// TwinCAT 3 PLC project Projekt
// ProgramVersion: 3.1.4023.0
// libraries:
//   Tc2_MC2, * (Beckhoff Automation GmbH)
//   Tc2_MC2_Camming, * (Beckhoff Automation GmbH)
//   Tc2_MC2_Drive, * (Beckhoff Automation GmbH)
//   Tc2_Standard, * (Beckhoff Automation GmbH)
//   Tc2_System, * (Beckhoff Automation GmbH)
//   Tc2_Utilities, * (Beckhoff Automation GmbH)
//   Tc3_Module, * (Beckhoff Automation GmbH)
// project tree:
//   GVLs/ IO.TcGVL
//   / PlcTask.TcTTO (not stored)
//   POUs/ FB_INICIALIZACIJA.TcPOU, MAIN.TcPOU, PRG_INIT.TcPOU
// real-time tasks:
//   TASK PlcTask: cycle T#10ms, priority 20, ADS port 350
// motion (NC):
//   TASK NC-Task 1 SAF: cycle T#2ms, priority 4, ADS port 501
//   TASK NC-Task 1 SVB: cycle T#10ms, priority 8, ADS port 511
//   AXIS SLAVE - AX5000 (id 1)
//     General: UnitName=°
//     Dynamic: Acceleration=5029.17, Deceleration=5029.17, Jerk=651703
//     Velo: RefSearch=38.8099189453125, RefSync=38.8099189453125, SlowManual=194.049594726563, FastManual=1164.29756835938, Fast=3880.99189453125, Maximum=3880.99
//     PositionAreaControl: Enable=false
//     TargetPosControl: Enable=false
//     OtherSettings: AllowMotionCmdToSlave=true
//     encoder EncType=8
//       EncPara: ScaleFactorNumerator=36, ScaleFactorDenominator=1048576, MaxCount=#xffffffff
//         Inc: RefSearchInverse=true, RefSyncInverse=false
//         TimeComp: TimeCompMode=1, EncDelayCycles=4
//     drive DrvType=9
//       DrvPara: MaxCount=#xffffffff, DriveControlDWord=#x00030100
//         Analog: VeloReferenz=4269.09108398438, VeloScale=1.02400649589962, TorqueSetpointScale=10, ScaleFactorActTorque=0.1
//         TimeComp: TaskDelayCycles=1
//     controller CtrType=1
//       CtrPara: PriorControlFactor=1
//         PosDiffControl: Enable=false
//         Observer: BandWidth=20
//   AXIS Enkoder_Axis (id 2)
//     General: UnitName=°, UnitFlags=#x00000004
//     Dynamic: AccelerationMaximum=25000, DecelerationMaximum=25000
//     Velo: Maximum=20000
//     PositionAreaControl: Enable=false
//     TargetPosControl: Enable=false
//     OtherSettings: AllowMotionCmdToSlave=true
//     encoder EncType=4
//       EncPara: ScaleFactorNumerator=1, MaxCount=#xffffffff
//         Inc: RefSoftSyncMask=#x0000ffff
//     drive DrvType=5
//       Analog: VeloReferenz=22000, TorqueSetpointScale=10, ScaleFactorActTorque=0.1
//       TimeComp: TaskDelayCycles=1
//     controller CtrType=1
//       CtrPara: PriorControlFactor=1
//         PosDiffControl: Enable=false
//         Observer: BandWidth=20
//   AXIS Axis 3 (id 3)
//     OtherSettings: AllowMotionCmdToSlave=true
//     encoder EncType=1
//     drive DrvType=5
//       Analog: TorqueSetpointScale=10, ScaleFactorActTorque=0.1
//       TimeComp: TaskDelayCycles=1
//     controller CtrType=1
//       CtrPara: PriorControlFactor=1
//         Observer: BandWidth=20
//   AXIS Axis 4 HENGSTLER (id 4)
//     General: UnitName=°, UnitFlags=#x00000004
//     OtherSettings: AllowMotionCmdToSlave=true
//     encoder EncType=5
//       EncPara: ScaleFactorNumerator=360, ScaleFactorDenominator=4096, ReferenceSystem=1
//     drive DrvType=5
//       Analog: TorqueSetpointScale=10, ScaleFactorActTorque=0.1
//       TimeComp: TaskDelayCycles=1
//     controller CtrType=1
//       CtrPara: PriorControlFactor=1
//         Observer: BandWidth=20
// I/O:
//   DEVICE Device 1 (EtherCAT), AmsNetId 5.67.218.26.2.1
//     Term 10 (EK1200) [EK1200-5000 EtherCAT Power supply (2A E-Bus)]
//       Term 10 (EL2252) [EL2252 2Ch. Dig. Output 24V, 0.5A, DC Time Stamp]
//       Term 11 (EL1252) [EL1252 2Ch. Fast Dig. Input 24V, 1µs, DC Latch]
//       Term 12 (EL2004) [EL2004 4Ch. Dig. Output 24V, 0.5A]
//       Term 13 (EL2004) [EL2004 4Ch. Dig. Output 24V, 0.5A]
//       Term 14 (EL1014) [EL1014 4Ch. Dig. Input 24V, 10µs]
//       Term 15 (EL5151-0021) [EL5151-0021 1Ch. Inc. Encoder, 24V DC Output]
//       Term 1 (EL5001) [EL5001 1Ch. SSI Encoder]
//       Term 17 (EL9011) [EL9011 End Terminal]
//   DEVICE Device 4 (EtherCAT), AmsNetId 5.67.218.26.5.1
//     Drive 8 (AX5106-0000-0214) [AX5106-0000-0214 EtherCAT Drive (SoE, 1 Ch.)]
//   DEVICE Device 2 (USB) (disabled)
//     Box 2 (C9900-L100 License-Key-USB-Stick)
// variable links:
//   NC-Task 1 SAF/Axes/Axis 4 HENGSTLER <-> Device 1 (EtherCAT)/Term 10 (EK1200)/Term 1 (EL5001)
//     Enc/Inputs/In/nDataIn1 <-> SSI Inputs/Counter value
//     Enc/Inputs/In/nState1 <-> SSI Inputs/Status/Data error
//     Enc/Inputs/In/nState1 @bit 1 <-> SSI Inputs/Status/Frame error
//     Enc/Inputs/In/nState1 @bit 2 <-> SSI Inputs/Status/Power failure
//     Enc/Inputs/In/nState2 @bit 5 <-> SSI Inputs/Status/Sync error
//     Enc/Inputs/In/nState4 @bit 1 <-> WcState/InputToggle
//     Enc/Inputs/In/nState4 <-> WcState/WcState
//   NC-Task 1 SAF/Axes/Enkoder_Axis <-> Device 1 (EtherCAT)/Term 10 (EK1200)/Term 15 (EL5151-0021)
//     Enc/Inputs/In/nDataIn1 <-> ENC Status/Counter value
//     Enc/Inputs/In/nDataIn2 <-> ENC Status/Latch value
//     Enc/Inputs/In/nState1 <-> ENC Status/Status/Latch C valid
//     Enc/Inputs/In/nState1 @bit 1 <-> ENC Status/Status/Latch extern valid
//     Enc/Inputs/In/nState1 @bit 2 <-> ENC Status/Status/Set counter done
//     Enc/Inputs/In/nState2 @bit 5 <-> ENC Status/Status/Compatible input cycle counter high
//     Enc/Inputs/In/nState2 @bit 4 <-> ENC Status/Status/Status of extern latch
//     Enc/Inputs/In/nState2 <-> ENC Status/Status/Status of input A
//     Enc/Inputs/In/nState2 @bit 1 <-> ENC Status/Status/Status of input B
//     Enc/Inputs/In/nState2 @bit 2 <-> ENC Status/Status/Status of input C
//     Enc/Inputs/In/nState2 @bit 7 <-> ENC Status/Status/TxPDO Toggle
//     Enc/Inputs/In/nState3 @bit 1 <-> ENC Status/Status/Measurement done
//     Enc/Inputs/In/nState3 <-> ENC Status/Status/Status of output
//     Enc/Inputs/In/nState4 @bit 1 <-> WcState/InputToggle
//     Enc/Inputs/In/nState4 <-> WcState/WcState
//     Enc/Outputs/Out/nCtrl1 <-> ENC Control/Control/Enable latch C
//     Enc/Outputs/Out/nCtrl1 @bit 3 <-> ENC Control/Control/Enable latch extern on negative edge
//     Enc/Outputs/Out/nCtrl1 @bit 1 <-> ENC Control/Control/Enable latch extern on positive edge
//     Enc/Outputs/Out/nCtrl1 @bit 6 <-> ENC Control/Control/Enable measurement
//     Enc/Outputs/Out/nCtrl1 @bit 5 <-> ENC Control/Control/Enable output functions
//     Enc/Outputs/Out/nCtrl1 @bit 2 <-> ENC Control/Control/Set counter
//     Enc/Outputs/Out/nCtrl1 @bit 7 <-> ENC Control/Control/Set counter on latch C
//     Enc/Outputs/Out/nCtrl1 @bit 4 <-> ENC Control/Control/Set output
//     Enc/Outputs/Out/nDataOut1 <-> ENC Control/Set counter value
//   NC-Task 1 SAF/Axes/SLAVE - AX5000 <-> Device 4 (EtherCAT)/Drive 8 (AX5106-0000-0214)
//     Drive/Inputs/In/nDataIn1 <-> AT/Following distance
//     Drive/Inputs/In/nDcOutputTime <-> InfoData/DcOutputShift
//     Drive/Inputs/In/nState1 <-> AT/Drive status word @bit 8
//     Drive/Inputs/In/nState2 <-> AT/Drive status word
//     Drive/Inputs/In/nState4 @bit 1 <-> WcState/InputToggle
//     Drive/Inputs/In/nState4 <-> WcState/WcState
//     Drive/Outputs/Out/nCtrl1 <-> MDT/Master control word @bit 8
//     Drive/Outputs/Out/nDataOut1 <-> MDT/Position command value
//     Enc/Inputs/In/nDataIn1 <-> AT/Position feedback 1 value
//     Enc/Inputs/In/nDcInputTime <-> InfoData/DcInputShift
//     Enc/Inputs/In/nState4 @bit 1 <-> WcState/InputToggle
//     Enc/Inputs/In/nState4 <-> WcState/WcState
//   Projekt/Projekt Instance <-> Device 1 (EtherCAT)/Term 10 (EK1200)/Term 11 (EL1252)
//     PlcTask Inputs/IO.bExternalCam <-> Channel 2/Input
//     PlcTask Inputs/IO.bZunanjiSignalTrigger <-> Channel 1/Input
//   Projekt/Projekt Instance <-> Device 1 (EtherCAT)/Term 10 (EK1200)/Term 12 (EL2004)
//     PlcTask Outputs/IO.bVklopIzpih <-> Channel 2/Output
//     PlcTask Outputs/IO.bVklopVakum <-> Channel 1/Output
//   Projekt/Projekt Instance <-> Device 1 (EtherCAT)/Term 10 (EK1200)/Term 14 (EL1014)
//     PlcTask Inputs/IO.bInit <-> Channel 4/Input
//     PlcTask Inputs/IO.bVakumOK <-> Channel 1/Input
//   Projekt/Projekt Instance <-> NC-Task 1 SAF/Axes/Axis 4 HENGSTLER
//     PlcTask Inputs/MAIN.MASTERENCODER.NcToPlc <-> Outputs/ToPlc
//     PlcTask Inputs/MAIN.r_MasterAngle <-> Outputs/ToPlc/ModuloActPos
//     PlcTask Outputs/MAIN.MASTERENCODER.PlcToNc <-> Inputs/FromPlc
//   Projekt/Projekt Instance <-> NC-Task 1 SAF/Axes/Enkoder_Axis
//     PlcTask Inputs/MAIN.MASTERAXIS.NcToPlc <-> Outputs/ToPlc
//     PlcTask Inputs/MAIN.realAngle <-> Outputs/ToPlc/ModuloActPos
//     PlcTask Inputs/MAIN.u_MasterEncoderValue <-> Enc/Outputs/Out/nDataOut1[0]
//     PlcTask Outputs/MAIN.MASTERAXIS.PlcToNc <-> Inputs/FromPlc
//   Projekt/Projekt Instance <-> NC-Task 1 SAF/Axes/SLAVE - AX5000
//     PlcTask Inputs/MAIN.SLAVEAXIS.NcToPlc <-> Outputs/ToPlc
//     PlcTask Inputs/MAIN.rAX5000Modulo <-> Outputs/ToPlc/ModuloActPos
//     PlcTask Inputs/MAIN.rMasterAngle <-> Outputs/ToPlc/ActPos
//     PlcTask Outputs/MAIN.SLAVEAXIS.PlcToNc <-> Inputs/FromPlc

// ---- GVLs/IO.TcGVL
{attribute 'qualified_only'}
VAR_GLOBAL
	//INPUTS
	///EL1252 DI0 - bzunanji triger
	//		 DI1 - vakum OK	
	bZunanjiSignalTrigger AT %I* : BOOL;
	bVakumOK AT %I* : BOOL;
	bExternalCam AT %I* : BOOL;
	bInit AT %I* : BOOL;
	
	
	//OUTPUTS
		//EL2004
	// Q0 - vakum
	// Q1 - izpih
	bVklopVakum AT %Q* : BOOL;
	bVklopIzpih AT %Q* : BOOL;
	
	bVklopTekociTrak AT %Q* : BOOL;
	bSistemOK AT %Q* : BOOL;
	

END_VAR

// ---- POUs/FB_INICIALIZACIJA.TcPOU
FUNCTION_BLOCK FB_INICIALIZACIJA
VAR_INPUT
	b_SignalToTrig : BOOL;	
	i_nKorak : INT;
END_VAR
VAR_OUTPUT
	b_GibVIzhodisce : BOOL;
	b_GibVPozicijoCakanjaKosa : BOOL;
END_VAR
VAR
	initEdge: INT;
	CLK: INT;
	korak: INT;
	Q: INT;
	R_initEdge : R_TRIG;
	
END_VAR

//ob pritisku na Init tipko gre v izhodisce
R_initEdge(CLK:=b_SignalToTrig);


CASE korak OF
	0:
		IF R_initEdge.Q AND (i_nKorak <> 50) THEN
		main.iKorak := -1;
		END_IF;
		korak := 10;
	10:
		
		IF (main.iKorak = 50) AND R_initEdge.Q THEN	
			main.iKorakRelativnegaPomika := -1;
		END_IF
	
		IF main.iKorak = 100 THEN
			korak := 0;
		END_IF
	
END_CASE

END_FUNCTION_BLOCK

// ---- POUs/MAIN.TcPOU
PROGRAM MAIN
VAR
	nCounterValue AT %I* : UINT;
	nCOunter1551 AT %I* : UDINT;
	
	// CAM
	MASTERAXIS : AXIS_REF;
	SLAVEAXIS :AXIS_REF;
	MASTERENCODER: AXIS_REF;
	
	adsadd AT%I* : T_AmsNetIdArr;
	
	//NC - POWER
	fbMaster_Power : MC_POWER;
	fbSlave_Power : MC_POWER;
	//NC - RESET
	fbMaster_Reset : MC_Reset;
	fbSlave_Reset : MC_Reset;
	fbSoeSlave_Reset : FB_SoEReset;
	
	iKorak : INT := 100;
	//NC - RESET AXIS
	
	//NC CAM IN&OUT
	fbCamIn : MC_CamIn;
	fbCamOut : MC_CamOut;
	//NC CAM OUT
	bCAMin : BOOL := FALSE;
	bResetMaster : BOOL;
	bResetSlave : BOOL;
	bPowerMaster : BOOL;
	bPowerSlave : BOOL;
	
	//
	fbSlaveMoveAbsolute : MC_MoveAbsolute;
	fbSlaveMoveRelative : MC_MoveRelative;
	fbSlaveMoveRelative2 : MC_MoveRelative;
	
	bMasterAbsoluteMove: BOOL := FALSE;
	
	rMasterAngle AT %I* : LREAL ;

	bSlaveMoveAbsolute : BOOL;
	bCAMOut: BOOL;
	
	u_MasterEncoderValue AT %I* : UINT;
	r_MasterAngle AT %I*: LREAL;
	
	bSlaveMoveRelative: BOOL;
	bMoveRelative : BOOL;
	SlaveDistance: LREAL;
	iKorakRelativnegaPomika: INT;
	SlaveRelativeSPeed: LREAL := 720;
	
	
	//SLAVE ABSOLUTE POSTIION
	rZeroAbsolutePosition : LREAL := 0;
	
	SlaveAbsoluteValue: LREAL;
	redgeTrigg : R_TRIG;
	PulzeQ1: TP;
	PulzeQ2: TP;
	bVakumON: BOOL;
	bIzpihON: BOOL;
	
	realAngle AT %I*: LREAL;
	
	SlaveHomming : MC_HOME;
	
	goHome: BOOL;
	
	rAX5000Modulo AT %I* : LREAL;
	
	bManualTurnOnIzpih: BOOL;
	
	b_error : BOOL;
	b_errorNiIzdelkaNaPrijemalu: BOOL;
	b_errorManipulatorNeinicializiran : BOOL;
	b_AX500_ch1_reset: BOOL;
	
	kotvkotu : R_TRIG;
	kotvkotu2 : R_TRIG;
	initEdge: R_TRIG;
	
	bSistemVNacinuRocno: BOOL;
	bSlaveMoveRelative2: BOOL;
	SlaveDistance2: LREAL;
END_VAR

VAR RETAIN PERSISTENT
	aktivacija2tockovnegaizvzema: BOOL;
	iCamCableID : INT;
	init : INT;
END_VAR


redgeTrigg(CLK:=io.bZunanjiSignalTrigger);
//kotvkotu(CLK:=r_MasterAngle > 259);
//kotvkotu2(CLK:=r_MasterAngle > 259);

kotvkotu(CLK:=r_MasterAngle > 120);
kotvkotu2(CLK:=r_MasterAngle > 270);


fbCamOut(Slave := SLAVEAXIS,
			Execute := bCAMOut);
			
fbMaster_Reset(Axis:=MASTERAXIS,
					Execute := bResetMaster);
					
fbSlave_Reset(Axis:=SLAVEAXIS,
					Execute := bResetSlave);

SLAVEAXIS.DriveAddress.NetID := F_CreateAmsNetId(nIds:= adsadd);
					
fbSoeSlave_Reset(Axis:=SLAVEAXIS, NetId := SLAVEAXIS.DriveAddress.NetID , Execute :=b_AX500_ch1_reset, Timeout := T#10S );	



fbMaster_Power (Axis := MASTERAXIS,
					Enable := bPowerMaster,
					Enable_Positive := TRUE,
					Enable_Negative := TRUE,
					Override := 100);
					
fbSlave_Power (Axis := SLAVEAXIS,
					Enable := bPowerSlave,
					Enable_Positive := TRUE,
					Enable_Negative := TRUE,
					Override := 100);	

 fbSlaveMoveAbsolute(Axis:=SLAVEAXIS, 
						Execute := bSlaveMoveAbsolute, 
						Position := SlaveAbsoluteValue, 
						Velocity := 360, 
						Acceleration := 4000, 
						Deceleration := 4000,
						Jerk := 0
						);	


fbSlaveMoveRelative(Axis:=SLAVEAXIS,
					Execute := bSlaveMoveRelative,
					Distance := SlaveDistance,
					Velocity := 1300, 
					Acceleration := 10000, 
					Deceleration := 10000,
					Jerk := 0,
					BufferMode :=MC_BufferMode.MC_BlendingLow);
					
fbSlaveMoveRelative2(
	Axis:=SLAVEAXIS , 
	Execute:= bSlaveMoveRelative2 , 
	Distance:=SlaveDistance2 , 
	Velocity:=1200 , 
	Acceleration:=9000 , 
	Deceleration:=9000, 
	Jerk:=0 , 
	BufferMode:= MC_BufferMode.MC_BlendingLow , 
	Options:= , 
	Done=> , 
	Busy=> , 
	Active=> , 
	CommandAborted=> , 
	Error=> , 
	ErrorID=> );
						
fbCamIn(Master:=MASTERENCODER,Slave:=SLAVEAXIS,Execute:=bCAMIN, CamTableID :=iCamCableID,SlaveOffset := 0);


			
CASE iKorak OF 
	-1:
	iKorakRelativnegaPomika := 100;
	bSlaveMoveAbsolute := FALSE;
	bCAMOut := TRUE;
	iKorak:=10;
	goHome := FALSE;
	
	b_errorNiIzdelkaNaPrijemalu := FALSE;
	
	aktivacija2tockovnegaizvzema := FALSE;
	bSistemVNacinuRocno := FALSE;
	//VAKUM IN IZPIH 
	bVakumON := TRUE;
	bManualTurnOnIzpih := FALSE;
	//
	10:
	bCAMOut := FALSE;
	iKorak := 20;
	
	20://RESET ERROR
	bResetMaster := TRUE;
	bResetSlave := TRUE;
	
	IF fbMaster_Reset.Done AND fbSlave_Reset.done THEN
		bResetMaster := FALSE;
		bResetSlave := FALSE;
		
		iKorak := 30;	
	END_IF;
					
	//iKorak := 30;
	30://VKLOP MOTORJA				
	
	
	IF NOT fbMaster_Power.ERROR AND NOT fbSlave_Power.ERROR THEN
		bPowerMaster := TRUE;
		bPowerSlave := TRUE;
		
		goHome := TRUE;
		
		IF SlaveHomming.Done THEN
			iKorak := 40;
		END_IF
	END_IF;
					
	//iKorak := 40;
	//40:
	
	
	40:
	  SlaveAbsoluteValue := 0;
	  bSlaveMoveAbsolute := TRUE; 
	  
	 IF fbSlaveMoveAbsolute.Done THEN
		
		 bSlaveMoveAbsolute := FALSE;
		 ikorak := 50; 
	 END_IF
	 //bMasterAbsoluteMove := FALSE;
	 45:
	 	SlaveDistance := 30;
		bSlaveMoveRelative := TRUE;
		
		IF fbSlaveMoveRelative.Done THEN
			bSlaveMoveRelative := FALSE;
			ikorak := 50;
		END_IF
	 50:
	 bMasterAbsoluteMove := FALSE;
	 
	 //skok na drugi progra
	
	 IF aktivacija2tockovnegaizvzema THEN
		 iKorakRelativnegaPomika := -1;
	 END_IF
	 
	 
		IF r_MasterAngle > 0 AND r_MasterAngle < 40  AND FALSE THEN
		bCAMIN := TRUE;
		  IF  fbCamIn.InSync THEN
		  ikorak := 60;
		  bCAMIN := FALSE;
		  END_IF
		END_IF
  
		  
	 
	 60:
	 // VKLOP IZPIHOVANJA
	 IF (r_MasterAngle > 155 AND r_MasterAngle < 355)  THEN
		 bVakumON := FALSE;
     ELSIF  r_MasterAngle < 5 THEN
		 bVakumON := TRUE;
		 bManualTurnOnIzpih := TRUE;
	 ELSE
		 bVakumON := TRUE;
		 bManualTurnOnIzpih := FALSE;
	 END_IF
	 
	 IF NOT IO.bVakumOK AND (r_MasterAngle > 250 AND r_MasterAngle < 350) THEN
		 b_errorNiIzdelkaNaPrijemalu := TRUE;
 	ELSE
		b_errorNiIzdelkaNaPrijemalu := FALSE;
	 END_IF
	 

	 
END_CASE;


CASE iKorakRelativnegaPomika OF
	-1: //absolute move to 0
	iKorak := 100;
		//VAKUM IN IZPIH 
	bVakumON := TRUE;
	bManualTurnOnIzpih := FALSE;
	
	b_errorNiIzdelkaNaPrijemalu := FALSE;
	
	bSistemVNacinuRocno := TRUE;
	
	IF bSlaveMoveAbsolute THEN
		bSlaveMoveAbsolute := FALSE;
	ELSE
		SlaveAbsoluteValue :=rZeroAbsolutePosition;
 		bSlaveMoveAbsolute := TRUE;
	END_IF
	
	IF fbSlaveMoveAbsolute.Done THEN
		bSlaveMoveAbsolute := FALSE;
		iKorakRelativnegaPomika := -10;
	END_IF
	(*
	
	
	*)
	
	-10: //distance move to 150° - cakanje na komad
	IF bSlaveMoveRelative THEN 
		bSlaveMoveRelative := FALSE;
	ELSE
		SlaveDistance := 141;
		bSlaveMoveRelative := TRUE;	
	END_IF
	
	IF fbSlaveMoveRelative.Done THEN
		bSlaveMoveRelative := FALSE;	
		iKorakRelativnegaPomika := 5;
	END_IF
	
	5://move to 180ž
	
	IF bMoveRelative OR redgeTrigg.Q OR kotvkotu.Q THEN
		SlaveDistance := 30;
		bSlaveMoveRelative := TRUE;
		//bVakumON := FALSE;
		bVakumON := NOT  TRUE;
	END_IF;
	
(*	IF fbSlaveMoveRelative.Busy THEN
		bSlaveMoveRelative := FALSE;	
		iKorakRelativnegaPomika := 10;
	END_IF
	
	*)
	
	IF fbSlaveMoveRelative.Done THEN
		bSlaveMoveRelative := FALSE;	
		iKorakRelativnegaPomika := 10;
		
	END_IF
	
	10: //move to 0
	//
	IF kotvkotu2.Q THEN
		//********		
		//slavedistance := 150 + 180 := 330
		//SlaveDistance := 330;
		
		//+++++
		SlaveDistance := 180;
		
		bSlaveMoveRelative := TRUE;	
	END_IF
			

	IF fbSlaveMoveRelative.Done THEN //nalaganje kosov na trak
		bSlaveMoveRelative := FALSE;
		
		//**************
		//preskoci 20 -> kar na 5
		//iKorakRelativnegaPomika := 5;
		
		//++++++++++
		iKorakRelativnegaPomika := 20;
		
		
		//bVakumON := TRUE;
        bIzpihON := TRUE;
		bManualTurnOnIzpih:= TRUE;
		bVakumON := NOT FALSE;
	END_IF
	
	20:

	SlaveDistance := 150;
	bSlaveMoveRelative := TRUE;	
	bIzpihON := FALSE;	
	IF fbSlaveMoveRelative.Done THEN //pozicija za izvzemanje kosov
		bSlaveMoveRelative := FALSE;
		bMoveRelative := FALSE;
		iKorakRelativnegaPomika := 5;
				
	END_IF
	bManualTurnOnIzpih := FALSE;
	
END_CASE

	IF fbMaster_Power.ERROR AND fbSlave_Power.ERROR THEN
		bPowerMaster := FALSE;
		bPowerSlave := FALSE;
	END_IF;

//VAKUM IN IZPIHOVANJE V NACINU
IF bSistemVNacinuRocno  THEN
// VKLOP IZPIHOVANJA
	 IF (rAX5000Modulo > 145 AND rAX5000Modulo < 350)  THEN
		 bVakumON := FALSE;
     ELSIF  rAX5000Modulo < 20   THEN
		 bVakumON := TRUE;
		 bManualTurnOnIzpih := TRUE;
	 ELSE
		 bVakumON := TRUE;
		 bManualTurnOnIzpih := FALSE;
	 END_IF	
END_IF;	
IO.bVklopVakum :=  bVakumON ;//OR NOT(rAX5000Modulo>160);	
IO.bVklopIzpih := bManualTurnOnIzpih ;//OR (rAX5000Modulo<3.0);

//PulzeQ1(IN := bIzpihON, PT:= T#100MS, Q=>IO.bVklopIzpih);

SlaveHomming(Axis:=SLAVEAXIS,Execute:=goHome, Position := 47,HomingMode:=MC_HomingMode.MC_DefaultHoming, bCalibrationCam := IO.bExternalCam);
IF SlaveHomming.Done THEN
	goHome := FALSE;
END_IF



//PRG_INIT();
//ob pritisku na Init tipko gre v izhodisce
initEdge(CLK:=IO.bInit);


CASE init OF
	0:
		IF initEdge.Q AND (main.iKorak <> 50) THEN
		iKorak := -1;
		init := 10;
		END_IF;
		
	10:
		
		IF (main.iKorak = 50) AND initEdge.Q THEN	
			MAIN.iKorakRelativnegaPomika := -1;
		END_IF
	
		IF iKorakRelativnegaPomika = 5 THEN
			init := 0;
		END_IF
	
END_CASE

END_PROGRAM

// ---- POUs/PRG_INIT.TcPOU
PROGRAM PRG_INIT
VAR
	init: INT;
	initEdge : R_TRIG;
END_VAR

//ob pritisku na Init tipko gre v izhodisce
initEdge(CLK:=IO.bInit);


CASE init OF
	0:
		IF initEdge.Q AND (main.iKorak <> 50) THEN
		MAIN.iKorak := -1;
		
		END_IF;
		init := 10;
	10:
		
		IF (main.iKorak = 50) AND initEdge.Q THEN	
			MAIN.iKorakRelativnegaPomika := -1;
		END_IF
	
		IF main.iKorak = 100 THEN
			init := 0;
		END_IF
	
END_CASE

END_PROGRAM
